Fanuc KAREL source: ka00205.KL

-- PROVISIONAL review KL for V770-1; original PC SHA256 7582bede2052090fa09ca42ab15bf3396aca9fe6c845fc8e8721b1abdd6c940c
-- Incomplete behavior may be omitted. Consult companion uncertainty JSON. Do not deploy.
PROGRAM KA00205
%NOLOCKGROUP
-- UNRESOLVED_DECL SRC type=002013
-- UNRESOLVED_DECL DST type=002013
BEGIN
  -- UNRESOLVED_PC offsets 5-19; opcodes 22,22,1E
  -- UNRESOLVED_PC offsets 24-28; opcodes 7F
END KA00205
